Fanuc KAREL source: kt00404.KL

-- PROVISIONAL review KL for V770-1; original PC SHA256 3f85c02be2baa42e84f00dac342fc80d3e97f0e72838a49353422de3d655ec62
-- Incomplete behavior may be omitted. Consult companion uncertainty JSON. Do not deploy.
PROGRAM KT00404
%NOLOCKGROUP
VAR
  I1 : INTEGER
  OUT : BOOLEAN
-- UNRESOLVED_DECL H2 type=002017
BEGIN
  -- UNRESOLVED_PC offsets 5-16; opcodes 2E,23
  -- UNRESOLVED_PC offsets 21-35; opcodes 2E,22,9D,33,B4
  -- UNRESOLVED_PC offsets 40-62; opcodes 21,22,9D,33,B3,5B,23
  -- UNRESOLVED_PC offsets 67-71; opcodes 7F
END KT00404
